DATA_BLOCK "ST10_Flow24_LUnloadingTrans_iDB"
{ S7_Optimized_Access := 'TRUE' }
VERSION : 0.1
NON_RETAIN
// ATTRIBUTES
// AUTO_NUMBER = False
// BLOCK_NUMBER = 1094
// END_ATTRIBUTES
"ST10_Flow24_LUnloadingTrans"

BEGIN

END_DATA_BLOCK

